// Mitsubishi GX Works2 project: mitsu_SCADA_PLC_v6.1   PLC: FX1N/FX1NC

PROGRAM MAIN
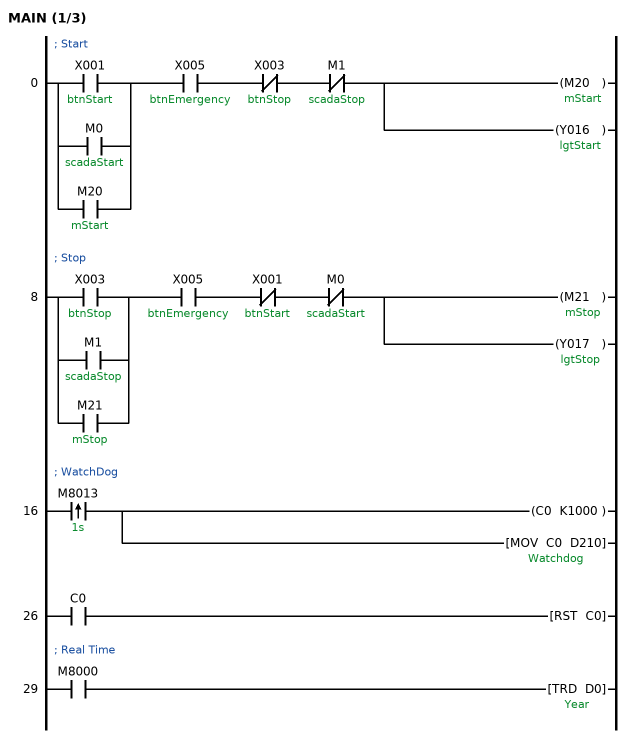
; Start
0     LD      X001  ; btnStart
      OR      M0  ; scadaStart
      OR      M20  ; mStart
      AND     X005  ; btnEmergency
      ANI     X003  ; btnStop
      ANI     M1  ; scadaStop
      OUT     M20  ; mStart
      OUT     Y016  ; lgtStart
; Stop
8     LD      X003  ; btnStop
      OR      M1  ; scadaStop
      OR      M21  ; mStop
      AND     X005  ; btnEmergency
      ANI     X001  ; btnStart
      ANI     M0  ; scadaStart
      OUT     M21  ; mStop
      OUT     Y017  ; lgtStop
; WatchDog
16    LDP     M8013  ; 1s
      OUT     C0 K1000
      MOV     C0 D210  ; Watchdog
26    LD      C0
      RST     C0
; Real Time
29    LD      M8000
      TRD     D0  ; Year
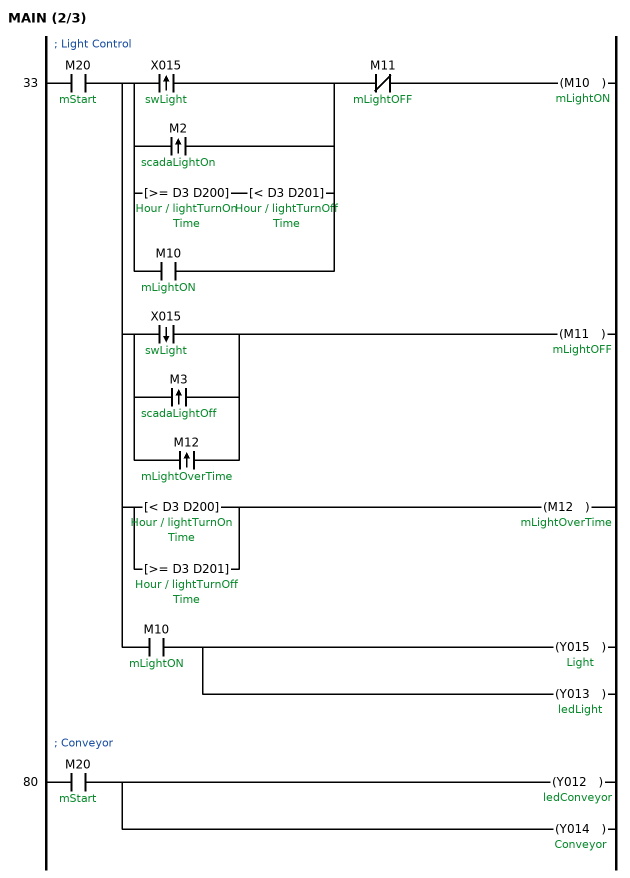
; Light Control
33    LD      M20  ; mStart
      MPS
      LDP     X015  ; swLight
      ORP     M2  ; scadaLightOn
      LD>=    D3 D200  ; Hour / lightTurnOnTime
      AND<    D3 D201  ; Hour / lightTurnOffTime
      ORB
      OR      M10  ; mLightON
      ANB
      ANI     M11  ; mLightOFF
      OUT     M10  ; mLightON
      MRD
      LDF     X015  ; swLight
      ORP     M3  ; scadaLightOff
      ORP     M12  ; mLightOverTime
      ANB
      OUT     M11  ; mLightOFF
      MRD
      LD<     D3 D200  ; Hour / lightTurnOnTime
      OR>=    D3 D201  ; Hour / lightTurnOffTime
      ANB
      OUT     M12  ; mLightOverTime
      MPP
      AND     M10  ; mLightON
      OUT     Y015  ; Light
      OUT     Y013  ; ledLight
; Conveyor
80    LD      M20  ; mStart
      OUT     Y012  ; ledConveyor
      OUT     Y014  ; Conveyor
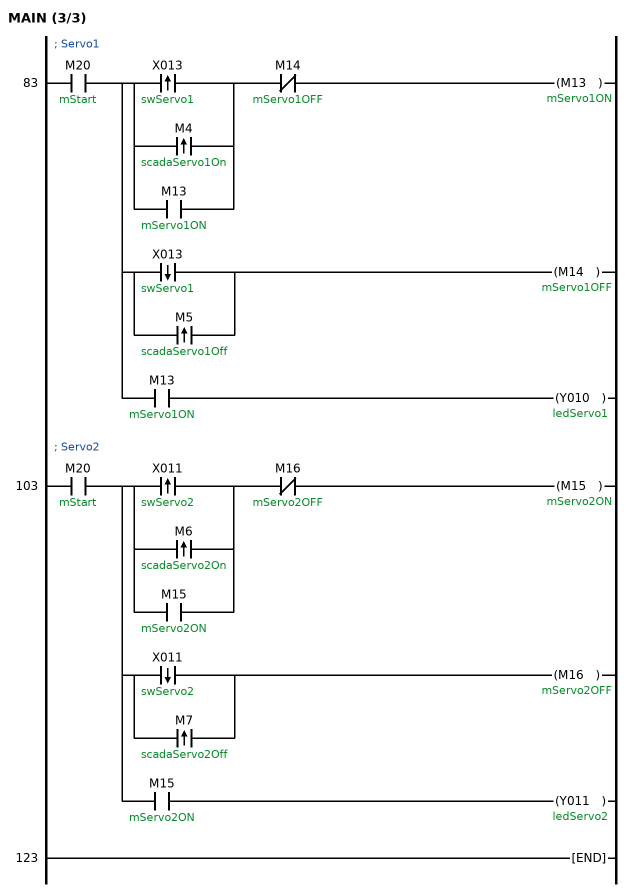
; Servo1
83    LD      M20  ; mStart
      MPS
      LDP     X013  ; swServo1
      ORP     M4  ; scadaServo1On
      OR      M13  ; mServo1ON
      ANB
      ANI     M14  ; mServo1OFF
      OUT     M13  ; mServo1ON
      MRD
      LDF     X013  ; swServo1
      ORP     M5  ; scadaServo1Off
      ANB
      OUT     M14  ; mServo1OFF
      MPP
      AND     M13  ; mServo1ON
      OUT     Y010  ; ledServo1
; Servo2
103   LD      M20  ; mStart
      MPS
      LDP     X011  ; swServo2
      ORP     M6  ; scadaServo2On
      OR      M15  ; mServo2ON
      ANB
      ANI     M16  ; mServo2OFF
      OUT     M15  ; mServo2ON
      MRD
      LDF     X011  ; swServo2
      ORP     M7  ; scadaServo2Off
      ANB
      OUT     M16  ; mServo2OFF
      MPP
      AND     M15  ; mServo2ON
      OUT     Y011  ; ledServo2
123   END
END_PROGRAM

// device comments not shown above
Y000  ; motorConveyor
Y001  ; servo1
Y002  ; servo2
M50  ; temp_0
M51  ; temp_1
M52  ; temp_2
M53  ; temp_3
M54  ; temp_4
M55  ; temp_5
D1  ; Month
D2  ; Day
D4  ; Minute
D5  ; Second
D6  ; Date
D202  ; temperature
